FUNCTION_BLOCK MSa (* Basic FB with empty ECC *)
  (* Standard: 61499-2 *)
  (* Version 1.0, 0000-00-00, 0 *)
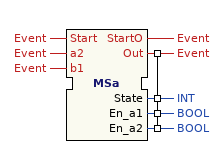
  EVENT_INPUT
    Start;
    a2;
    b1;
  END_EVENT
  EVENT_OUTPUT
    StartO;
    Out WITH State, En_a1, En_a2;
  END_EVENT
  VAR_OUTPUT
    State : INT := 1;
    En_a1 : BOOL := 1;
    En_a2 : BOOL := 1;
  END_VAR
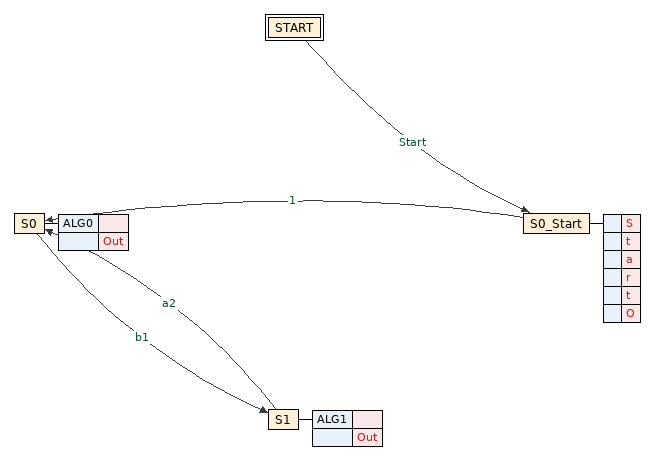
  EC_STATES
    START; (* Initial State *)
    S0_Start : -> S, -> t, -> a, -> r, -> t, -> O;
    S1 : ALG1, -> Out;
    S0 : ALG0, -> Out;
  END_STATES
  EC_TRANSITIONS
    START TO S0_Start := Start;
    S0_Start TO S0 := 1;
    S1 TO S0 := a2;
    S0 TO S1 := b1;
  END_TRANSITIONS
  ALGORITHM ALG1 IN ST:
State:=1;
				En_a1:=False;
				En_a2:=True;
  END_ALGORITHM
  ALGORITHM ALG0 IN ST:
State:=0;
				En_a1:=True;
				En_a2:=False;
  END_ALGORITHM
END_FUNCTION_BLOCK
